(* PLC project SafeLOGIC, BrAutomation SafeDESIGNER  5.24.1.0 *)
(* stored: companyURL http://www.br-automation.com, creationDateTime Fri Nov 28 14:24:40 2025 *)

PROGRAM Main
  VAR  (* added by the conversion: wires and edge detectors of the diagram *)
    _AND_S17_OUT : ANY;
    _AND_S38_OUT : SAFEBOOL;
  END_VAR

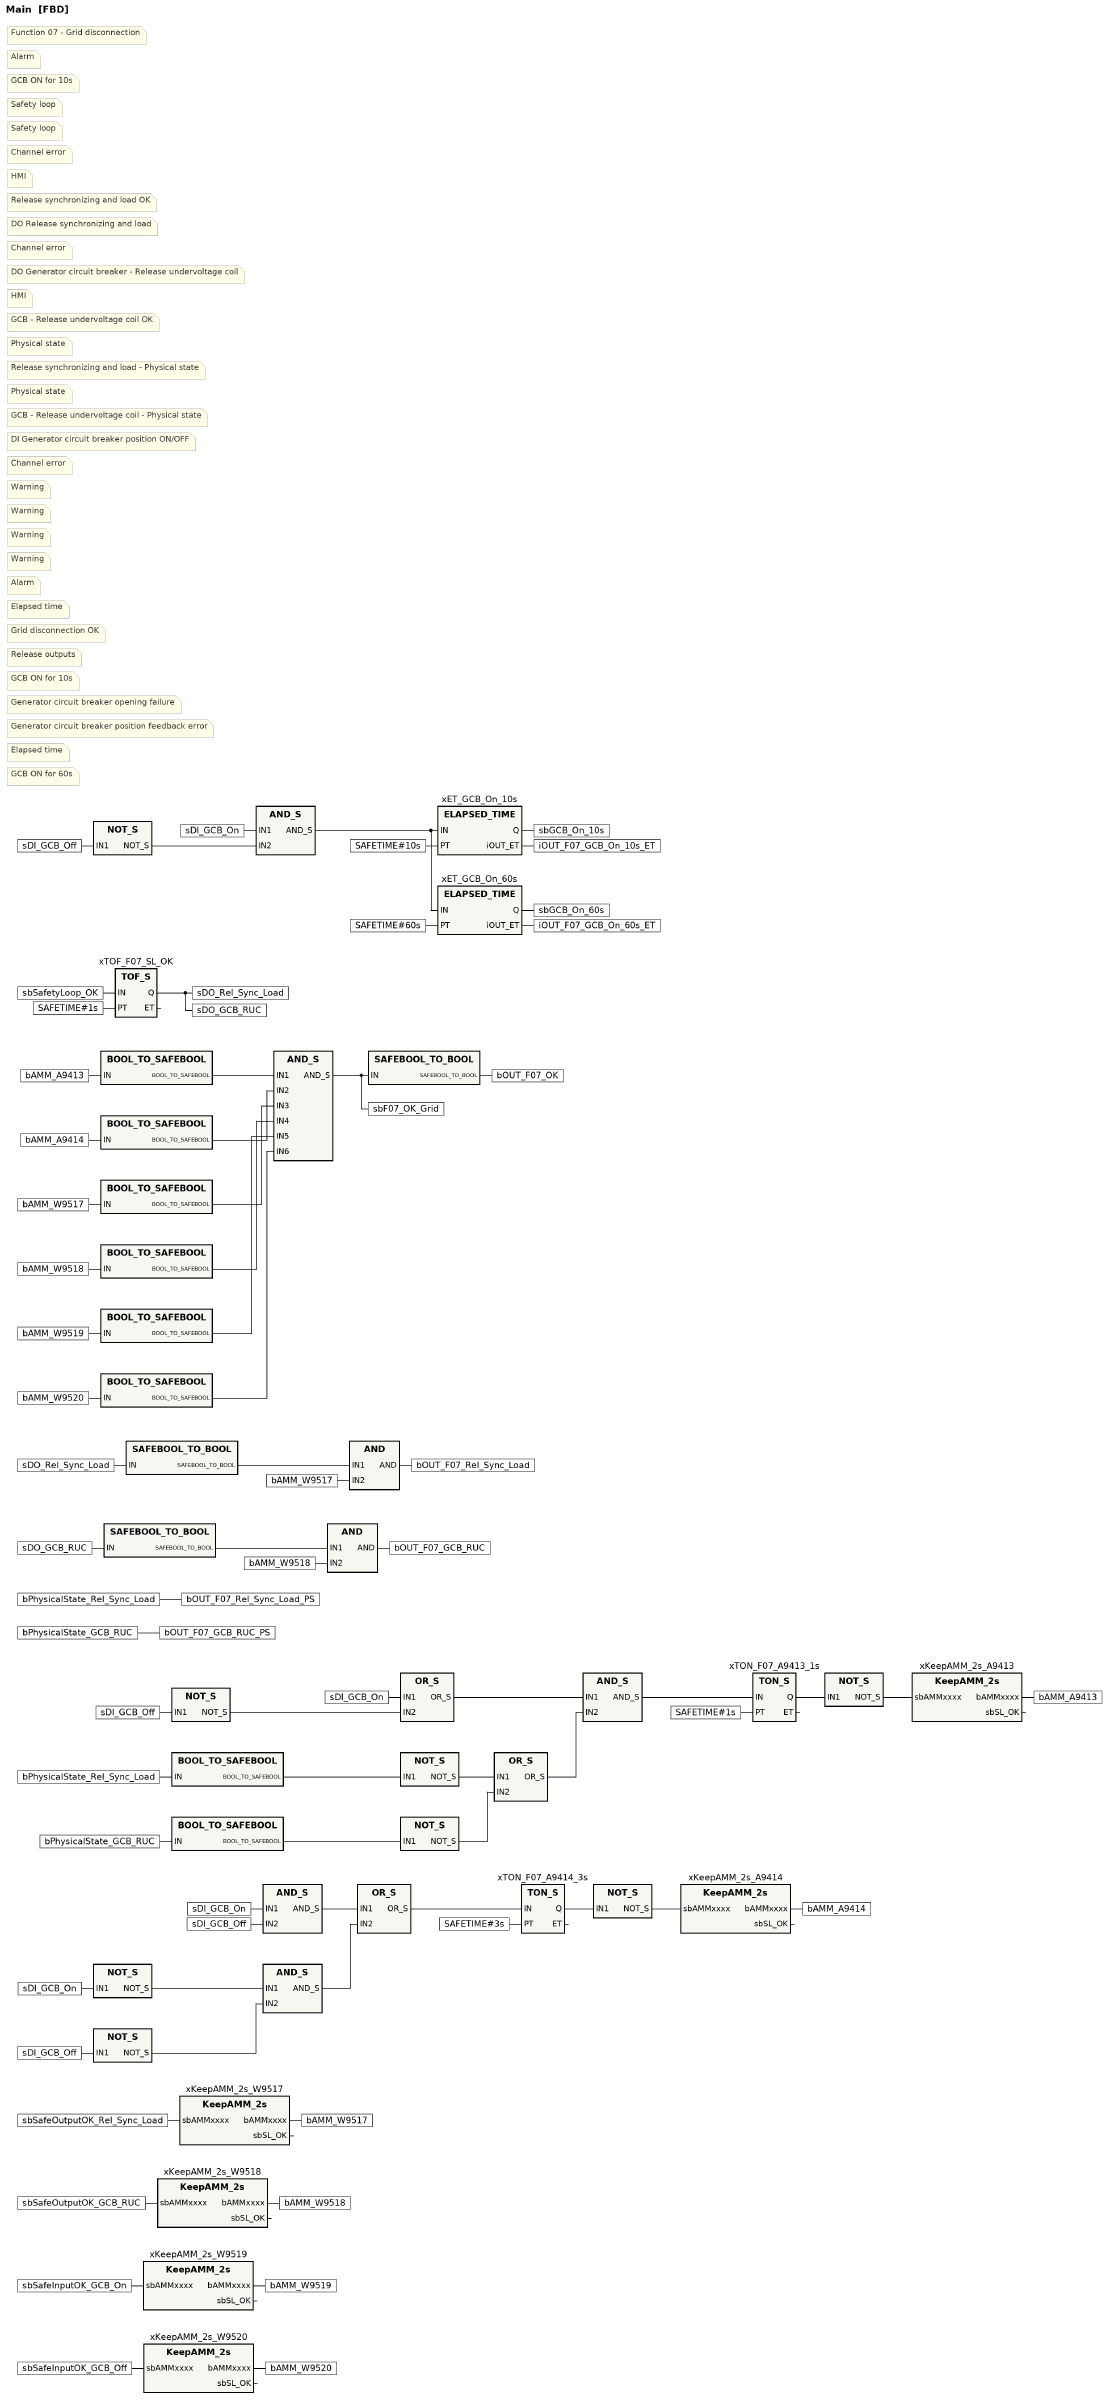
(* FBD diagram, written out as Structured Text *)
(* Function 07 - Grid disconnection *)
(* Release outputs *)
xTOF_F07_SL_OK(IN := sbSafetyLoop_OK, PT := SAFETIME#1s);
sDO_Rel_Sync_Load := xTOF_F07_SL_OK.Q;
sDO_GCB_RUC := xTOF_F07_SL_OK.Q;
(* DO Release synchronizing and load *)
(* Channel error *)
(* Warning *)
xKeepAMM_2s_W9517(sbAMMxxxx := sbSafeOutputOK_Rel_Sync_Load);
bAMM_W9517 := xKeepAMM_2s_W9517.bAMMxxxx;
(* HMI *)
(* Release synchronizing and load OK *)
bOUT_F07_Rel_Sync_Load := SAFEBOOL_TO_BOOL(sDO_Rel_Sync_Load) AND bAMM_W9517;
(* Physical state *)
(* Release synchronizing and load - Physical state *)
bOUT_F07_Rel_Sync_Load_PS := bPhysicalState_Rel_Sync_Load;
(* DO Generator circuit breaker - Release undervoltage coil *)
(* Channel error *)
(* Warning *)
xKeepAMM_2s_W9518(sbAMMxxxx := sbSafeOutputOK_GCB_RUC);
bAMM_W9518 := xKeepAMM_2s_W9518.bAMMxxxx;
(* HMI *)
(* GCB - Release undervoltage coil OK *)
bOUT_F07_GCB_RUC := SAFEBOOL_TO_BOOL(sDO_GCB_RUC) AND bAMM_W9518;
(* Physical state *)
(* GCB - Release undervoltage coil - Physical state *)
bOUT_F07_GCB_RUC_PS := bPhysicalState_GCB_RUC;
(* DI Generator circuit breaker position ON/OFF *)
(* Channel error *)
(* Warning *)
xKeepAMM_2s_W9519(sbAMMxxxx := sbSafeInputOK_GCB_On);
bAMM_W9519 := xKeepAMM_2s_W9519.bAMMxxxx;
(* Warning *)
xKeepAMM_2s_W9520(sbAMMxxxx := sbSafeInputOK_GCB_Off);
bAMM_W9520 := xKeepAMM_2s_W9520.bAMMxxxx;
(* Generator circuit breaker opening failure *)
(* Alarm *)
xTON_F07_A9413_1s(IN := AND_S(OR_S(sDI_GCB_On, NOT_S(sDI_GCB_Off)), OR_S(NOT_S(BOOL_TO_SAFEBOOL(bPhysicalState_Rel_Sync_Load)), NOT_S(BOOL_TO_SAFEBOOL(bPhysicalState_GCB_RUC)))), PT := SAFETIME#1s);
xKeepAMM_2s_A9413(sbAMMxxxx := NOT_S(xTON_F07_A9413_1s.Q));
bAMM_A9413 := xKeepAMM_2s_A9413.bAMMxxxx;
(* Generator circuit breaker position feedback error *)
(* Alarm *)
xTON_F07_A9414_3s(IN := OR_S(AND_S(sDI_GCB_On, sDI_GCB_Off), AND_S(NOT_S(sDI_GCB_On), NOT_S(sDI_GCB_Off))), PT := SAFETIME#3s);
xKeepAMM_2s_A9414(sbAMMxxxx := NOT_S(xTON_F07_A9414_3s.Q));
bAMM_A9414 := xKeepAMM_2s_A9414.bAMMxxxx;
(* GCB ON for 10s *)
(* GCB ON for 10s *)
(* Elapsed time *)
_AND_S17_OUT := AND_S(sDI_GCB_On, NOT_S(sDI_GCB_Off));
xET_GCB_On_10s(IN := _AND_S17_OUT, PT := SAFETIME#10s);
sbGCB_On_10s := xET_GCB_On_10s.Q;
iOUT_F07_GCB_On_10s_ET := xET_GCB_On_10s.iOUT_ET;
(* GCB ON for 60s *)
(* Elapsed time *)
xET_GCB_On_60s(IN := _AND_S17_OUT, PT := SAFETIME#60s);
sbGCB_On_60s := xET_GCB_On_60s.Q;
iOUT_F07_GCB_On_60s_ET := xET_GCB_On_60s.iOUT_ET;
(* Safety loop *)
(* Safety loop *)
(* Grid disconnection OK *)
_AND_S38_OUT := AND_S(BOOL_TO_SAFEBOOL(bAMM_A9413), BOOL_TO_SAFEBOOL(bAMM_A9414), BOOL_TO_SAFEBOOL(bAMM_W9517), BOOL_TO_SAFEBOOL(bAMM_W9518), BOOL_TO_SAFEBOOL(bAMM_W9519), BOOL_TO_SAFEBOOL(bAMM_W9520));
sbF07_OK_Grid := _AND_S38_OUT;
bOUT_F07_OK := SAFEBOOL_TO_BOOL(_AND_S38_OUT);
END_PROGRAM
